FUNCTION_BLOCK SS3_v_ps2 (* Composite FB wrapping other FBs *)
  (* Standard: 61499-2 *)
  (* Version 1.0, 2025-05-16, DEVIASH *)
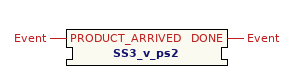
  EVENT_INPUT
    PRODUCT_ARRIVED;
  END_EVENT
  EVENT_OUTPUT
    DONE;
  END_EVENT
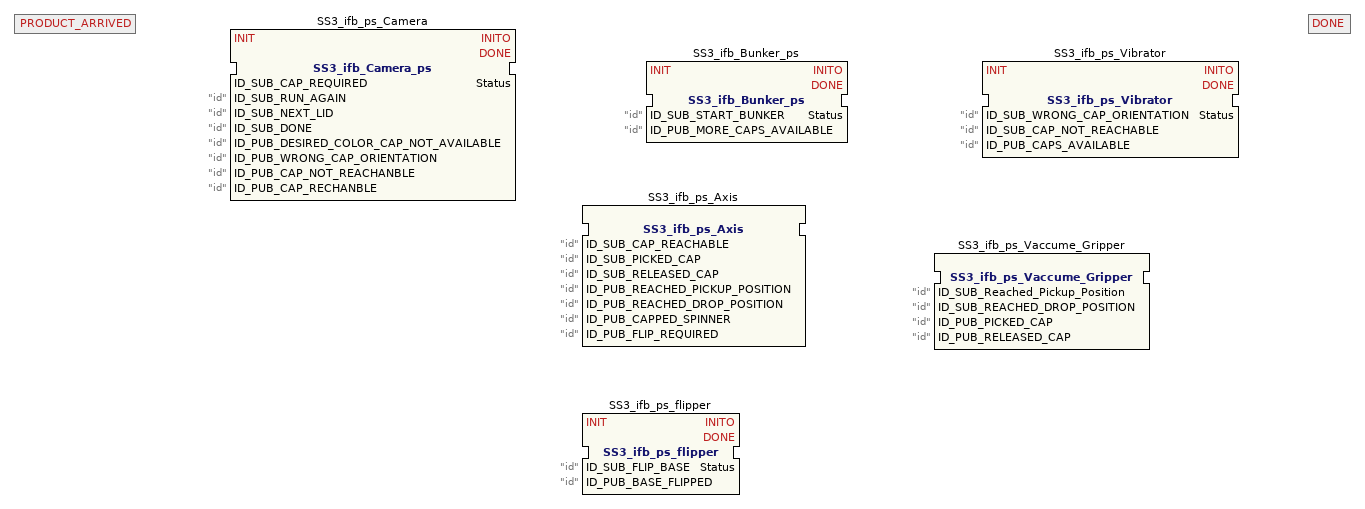
  FBS
    SS3_ifb_ps_Camera : SS3_ifb_Camera_ps(ID_SUB_RUN_AGAIN := "id", ID_SUB_NEXT_LID := "id", ID_SUB_DONE := "id", ID_PUB_DESIRED_COLOR_CAP_NOT_AVAILABLE := "id", ID_PUB_WRONG_CAP_ORIENTATION := "id", ID_PUB_CAP_NOT_REACHANBLE := "id", ID_PUB_CAP_RECHANBLE := "id");
    SS3_ifb_ps_Vaccume_Gripper : SS3_ifb_ps_Vaccume_Gripper(ID_SUB_Reached_Pickup_Position := "id", ID_SUB_REACHED_DROP_POSITION := "id", ID_PUB_PICKED_CAP := "id", ID_PUB_RELEASED_CAP := "id");
    SS3_ifb_ps_Vibrator : SS3_ifb_ps_Vibrator(ID_SUB_WRONG_CAP_ORIENTATION := "id", ID_SUB_CAP_NOT_REACHABLE := "id", ID_PUB_CAPS_AVAILABLE := "id");
    SS3_ifb_ps_flipper : SS3_ifb_ps_flipper(ID_SUB_FLIP_BASE := "id", ID_PUB_BASE_FLIPPED := "id");
    SS3_ifb_Bunker_ps : SS3_ifb_Bunker_ps(ID_SUB_START_BUNKER := "id", ID_PUB_MORE_CAPS_AVAILABLE := "id");
    SS3_ifb_ps_Axis : SS3_ifb_ps_Axis(ID_SUB_CAP_REACHABLE := "id", ID_SUB_PICKED_CAP := "id", ID_SUB_RELEASED_CAP := "id", ID_PUB_REACHED_PICKUP_POSITION := "id", ID_PUB_REACHED_DROP_POSITION := "id", ID_PUB_CAPPED_SPINNER := "id", ID_PUB_FLIP_REQUIRED := "id");
  END_FBS
END_FUNCTION_BLOCK
